// SIMATIC S7-200 project (STEP 7-Micro/WIN), CPU 224 CN REL 02.01

ORGANIZATION_BLOCK MAIN:OB1
TITLE=程序注释
BEGIN
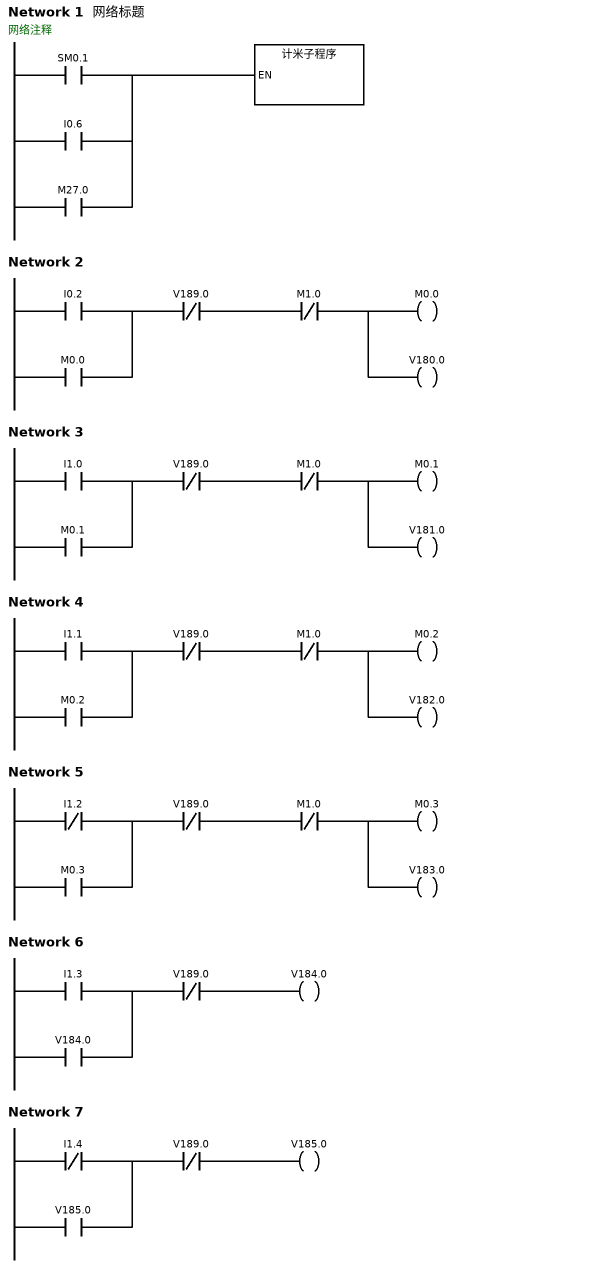
Network 1 // 网络标题
// 网络注释
LD     SM0.1
O      I0.6
O      M27.0
CALL   计米子程序:SBR0
Network 2
LD     I0.2
O      M0.0
AN     V189.0
AN     M1.0
=      M0.0
=      V180.0
Network 3
LD     I1.0
O      M0.1
AN     V189.0
AN     M1.0
=      M0.1
=      V181.0
Network 4
LD     I1.1
O      M0.2
AN     V189.0
AN     M1.0
=      M0.2
=      V182.0
Network 5
LDN    I1.2
O      M0.3
AN     V189.0
AN     M1.0
=      M0.3
=      V183.0
Network 6
LD     I1.3
O      V184.0
AN     V189.0
=      V184.0
Network 7
LDN    I1.4
O      V185.0
AN     V189.0
=      V185.0
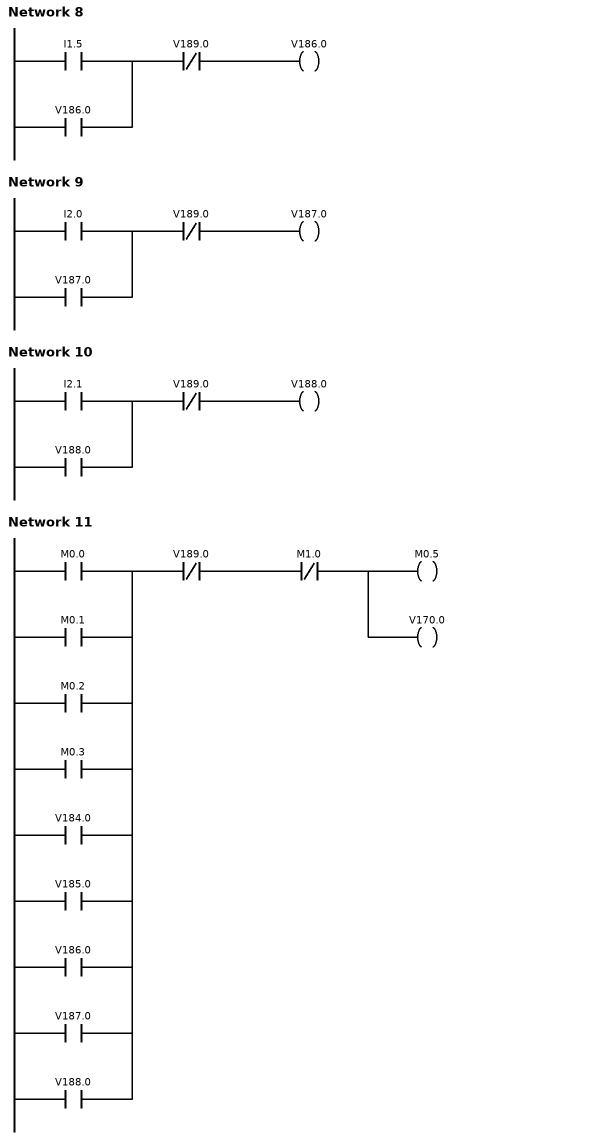
Network 8
LD     I1.5
O      V186.0
AN     V189.0
=      V186.0
Network 9
LD     I2.0
O      V187.0
AN     V189.0
=      V187.0
Network 10
LD     I2.1
O      V188.0
AN     V189.0
=      V188.0
Network 11
LD     M0.0
O      M0.1
O      M0.2
O      M0.3
O      V184.0
O      V185.0
O      V186.0
O      V187.0
O      V188.0
AN     V189.0
AN     M1.0
=      M0.5
=      V170.0
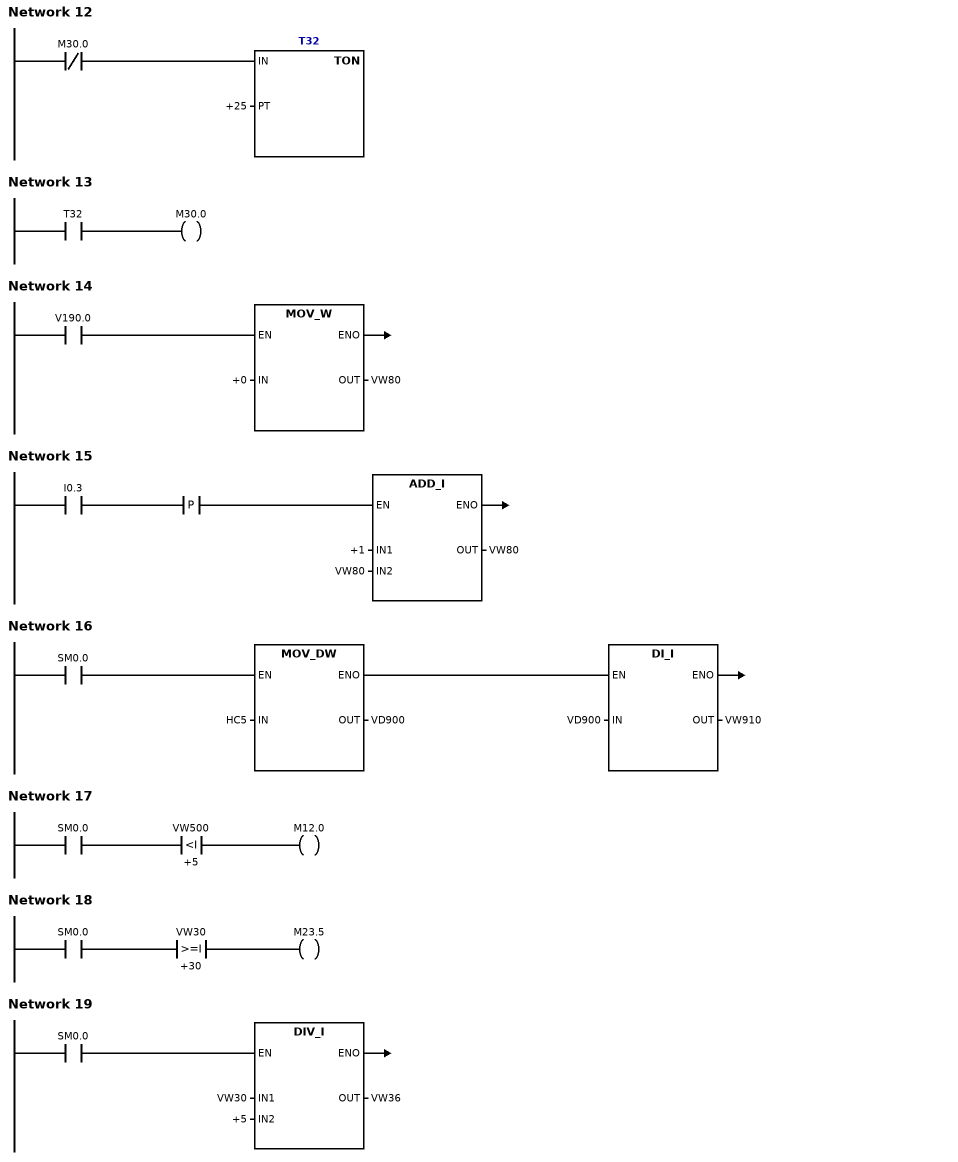
Network 12
LDN    M30.0
TON    T32, +25
Network 13
LD     T32
=      M30.0
Network 14
LD     V190.0
MOVW   +0, VW80
Network 15
LD     I0.3
EU
+I     +1, VW80
Network 16
LD     SM0.0
MOVD   HC5, VD900
AENO
DTI    VD900, VW910
Network 17
LD     SM0.0
AW<    VW500, +5
=      M12.0
Network 18
LD     SM0.0
AW>=   VW30, +30
=      M23.5
Network 19
LD     SM0.0
MOVW   VW30, VW36
/I     +5, VW36
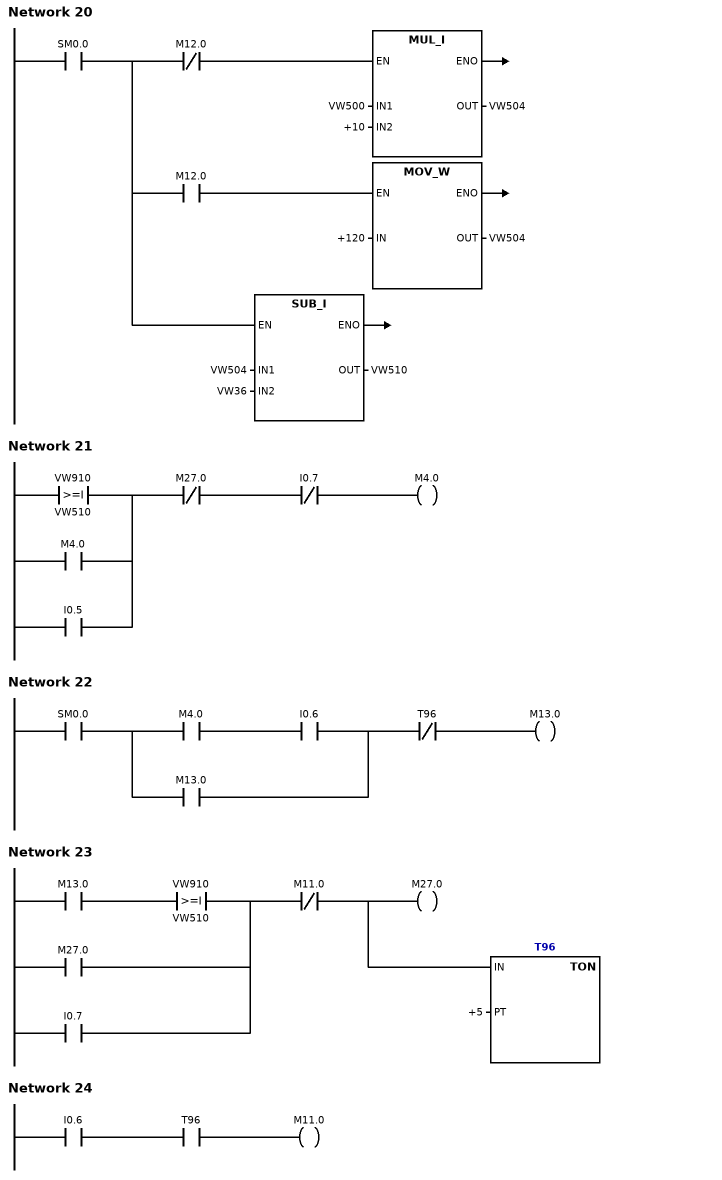
Network 20
LD     SM0.0
LPS
AN     M12.0
MOVW   VW500, VW504
*I     +10, VW504
LRD
A      M12.0
MOVW   +120, VW504
LPP
MOVW   VW504, VW510
-I     VW36, VW510
Network 21
LDW>=  VW910, VW510
O      M4.0
O      I0.5
AN     M27.0
AN     I0.7
=      M4.0
Network 22
LD     SM0.0
LD     M4.0
A      I0.6
O      M13.0
ALD
AN     T96
=      M13.0
Network 23
LD     M13.0
AW>=   VW910, VW510
O      M27.0
O      I0.7
AN     M11.0
=      M27.0
TON    T96, +5
Network 24
LD     I0.6
A      T96
=      M11.0
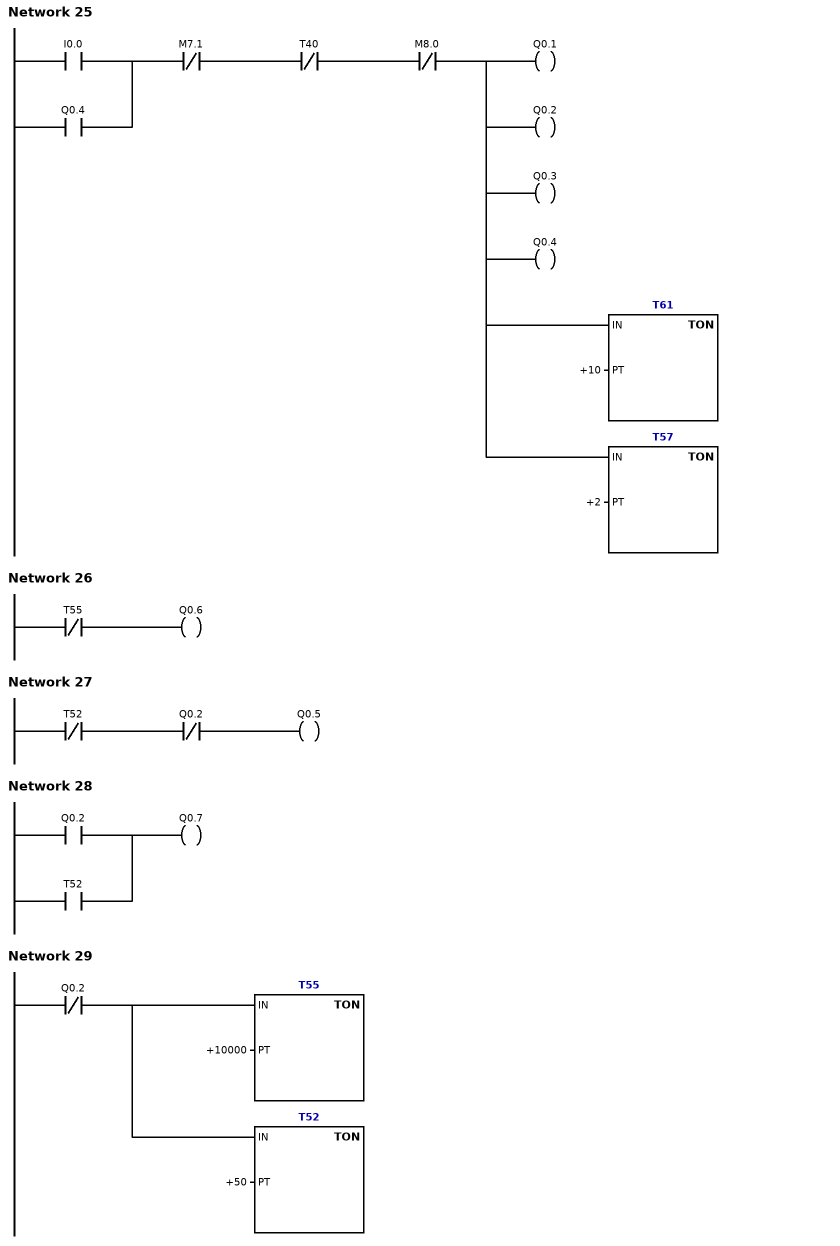
Network 25
LD     I0.0
O      Q0.4
AN     M7.1
AN     T40
AN     M8.0
=      Q0.1
=      Q0.2
=      Q0.3
=      Q0.4
TON    T61, +10
TON    T57, +2
Network 26
LDN    T55
=      Q0.6
Network 27
LDN    T52
AN     Q0.2
=      Q0.5
Network 28
LD     Q0.2
O      T52
=      Q0.7
Network 29
LDN    Q0.2
TON    T55, +10000
TON    T52, +50
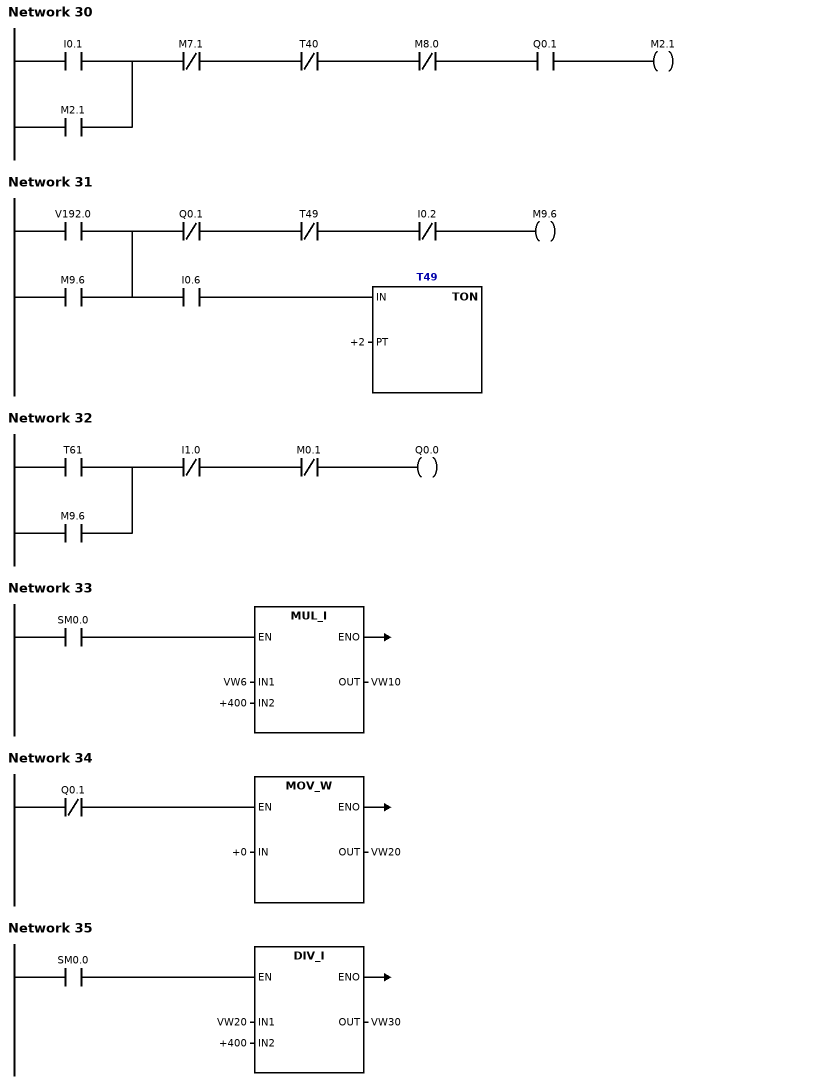
Network 30
LD     I0.1
O      M2.1
AN     M7.1
AN     T40
AN     M8.0
A      Q0.1
=      M2.1
Network 31
LD     V192.0
O      M9.6
LPS
AN     Q0.1
AN     T49
AN     I0.2
=      M9.6
LPP
A      I0.6
TON    T49, +2
Network 32
LD     T61
O      M9.6
AN     I1.0
AN     M0.1
=      Q0.0
Network 33
LD     SM0.0
MOVW   VW6, VW10
*I     +400, VW10
Network 34
LDN    Q0.1
MOVW   +0, VW20
Network 35
LD     SM0.0
MOVW   VW20, VW30
/I     +400, VW30
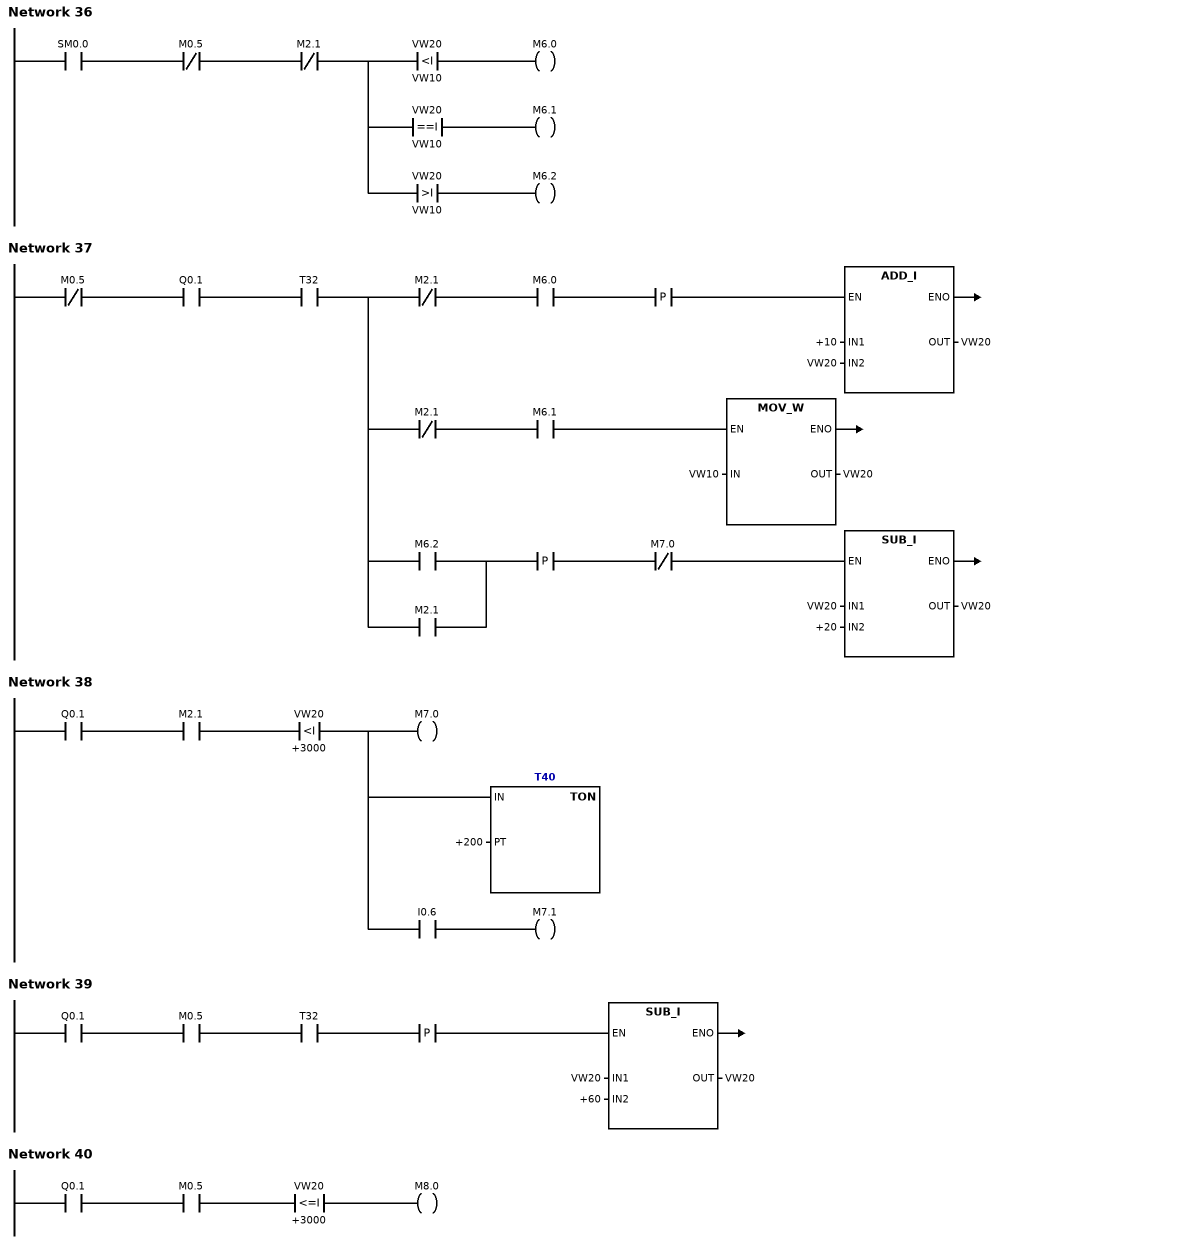
Network 36
LD     SM0.0
AN     M0.5
AN     M2.1
LPS
AW<    VW20, VW10
=      M6.0
LRD
AW=    VW20, VW10
=      M6.1
LPP
AW>    VW20, VW10
=      M6.2
Network 37
LDN    M0.5
A      Q0.1
A      T32
LPS
AN     M2.1
A      M6.0
EU
+I     +10, VW20
LRD
AN     M2.1
A      M6.1
MOVW   VW10, VW20
LPP
LD     M6.2
O      M2.1
ALD
EU
AN     M7.0
-I     +20, VW20
Network 38
LD     Q0.1
A      M2.1
AW<    VW20, +3000
=      M7.0
TON    T40, +200
A      I0.6
=      M7.1
Network 39
LD     Q0.1
A      M0.5
A      T32
EU
-I     +60, VW20
Network 40
LD     Q0.1
A      M0.5
AW<=   VW20, +3000
=      M8.0
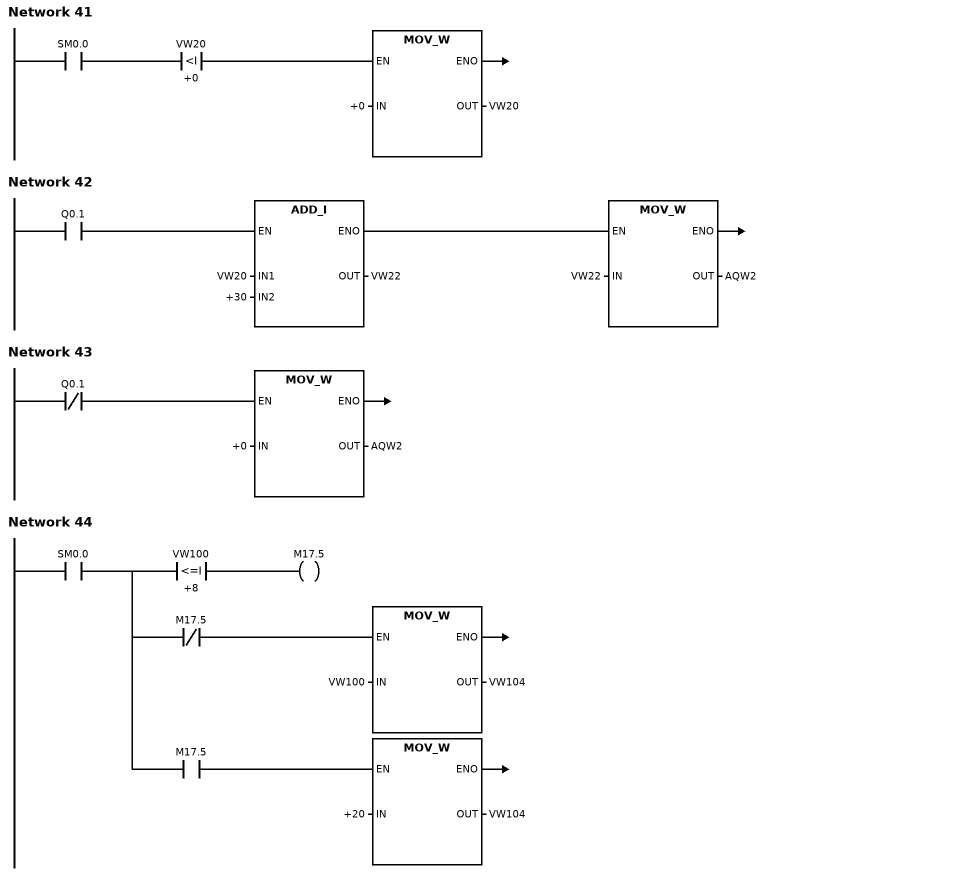
Network 41
LD     SM0.0
AW<    VW20, +0
MOVW   +0, VW20
Network 42
LD     Q0.1
MOVW   VW20, VW22
AENO
+I     +30, VW22
AENO
MOVW   VW22, AQW2
Network 43
LDN    Q0.1
MOVW   +0, AQW2
Network 44
LD     SM0.0
LPS
AW<=   VW100, +8
=      M17.5
LRD
AN     M17.5
MOVW   VW100, VW104
LPP
A      M17.5
MOVW   +20, VW104
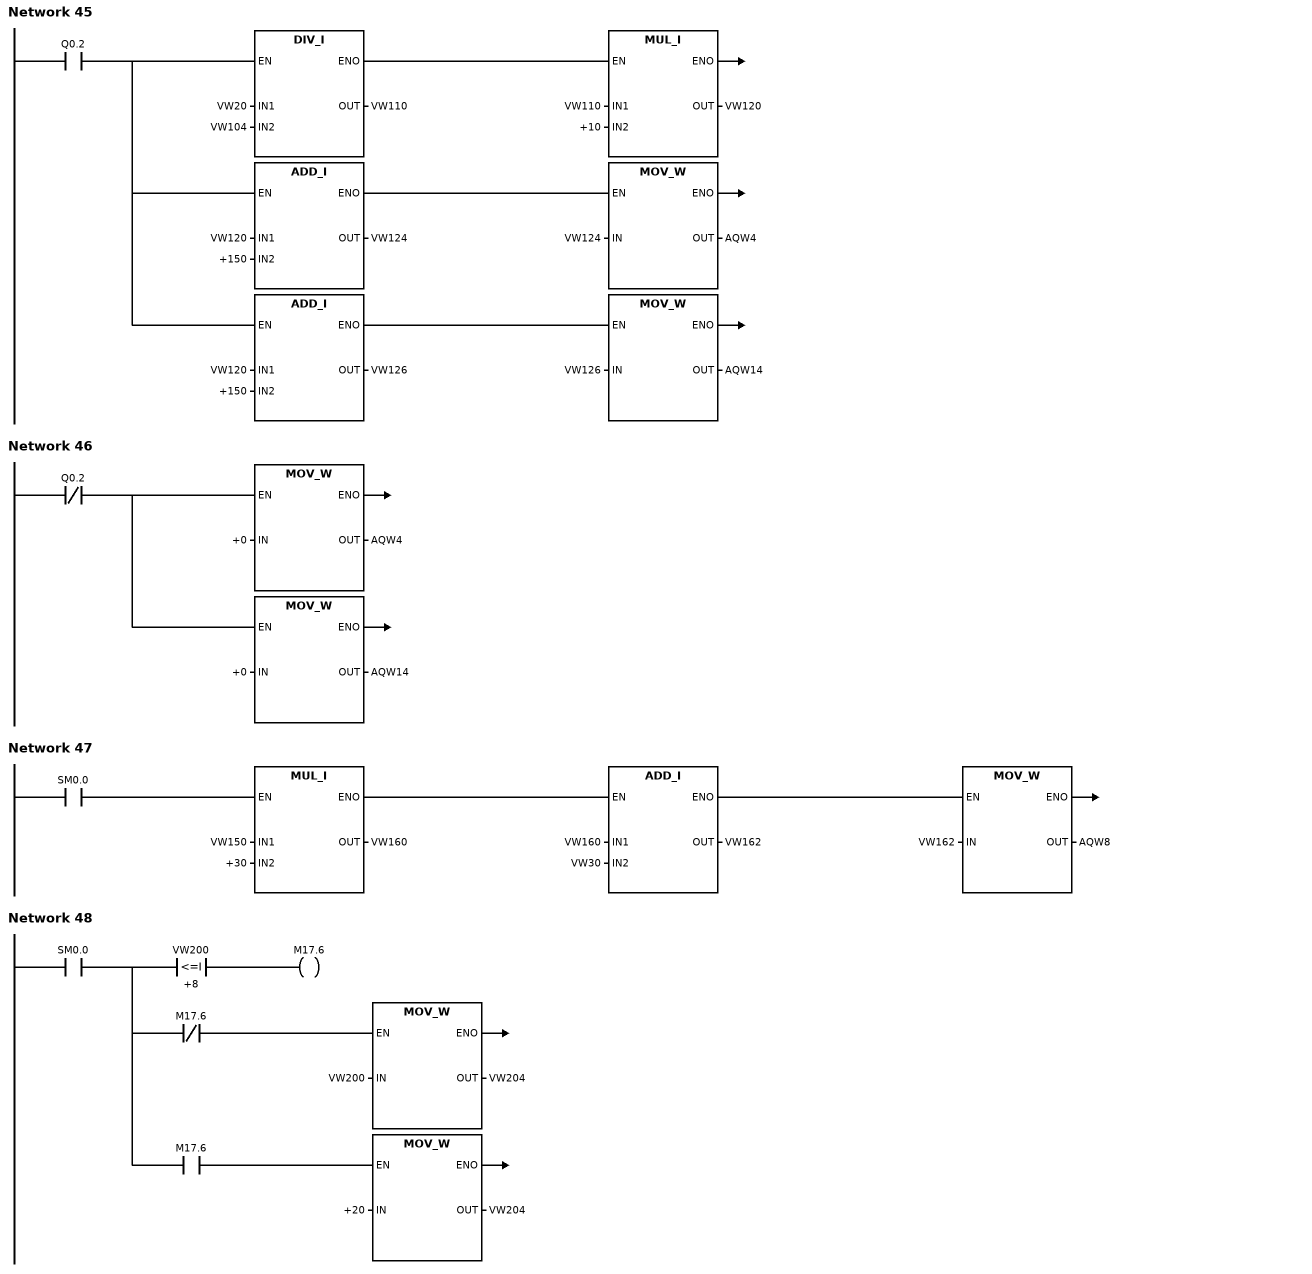
Network 45
LD     Q0.2
LPS
MOVW   VW20, VW110
AENO
/I     VW104, VW110
AENO
MOVW   VW110, VW120
*I     +10, VW120
LRD
MOVW   VW120, VW124
AENO
+I     +150, VW124
AENO
MOVW   VW124, AQW4
LPP
MOVW   VW120, VW126
AENO
+I     +150, VW126
AENO
MOVW   VW126, AQW14
Network 46
LDN    Q0.2
MOVW   +0, AQW4
MOVW   +0, AQW14
Network 47
LD     SM0.0
MOVW   VW150, VW160
AENO
*I     +30, VW160
AENO
MOVW   VW160, VW162
AENO
+I     VW30, VW162
AENO
MOVW   VW162, AQW8
Network 48
LD     SM0.0
LPS
AW<=   VW200, +8
=      M17.6
LRD
AN     M17.6
MOVW   VW200, VW204
LPP
A      M17.6
MOVW   +20, VW204
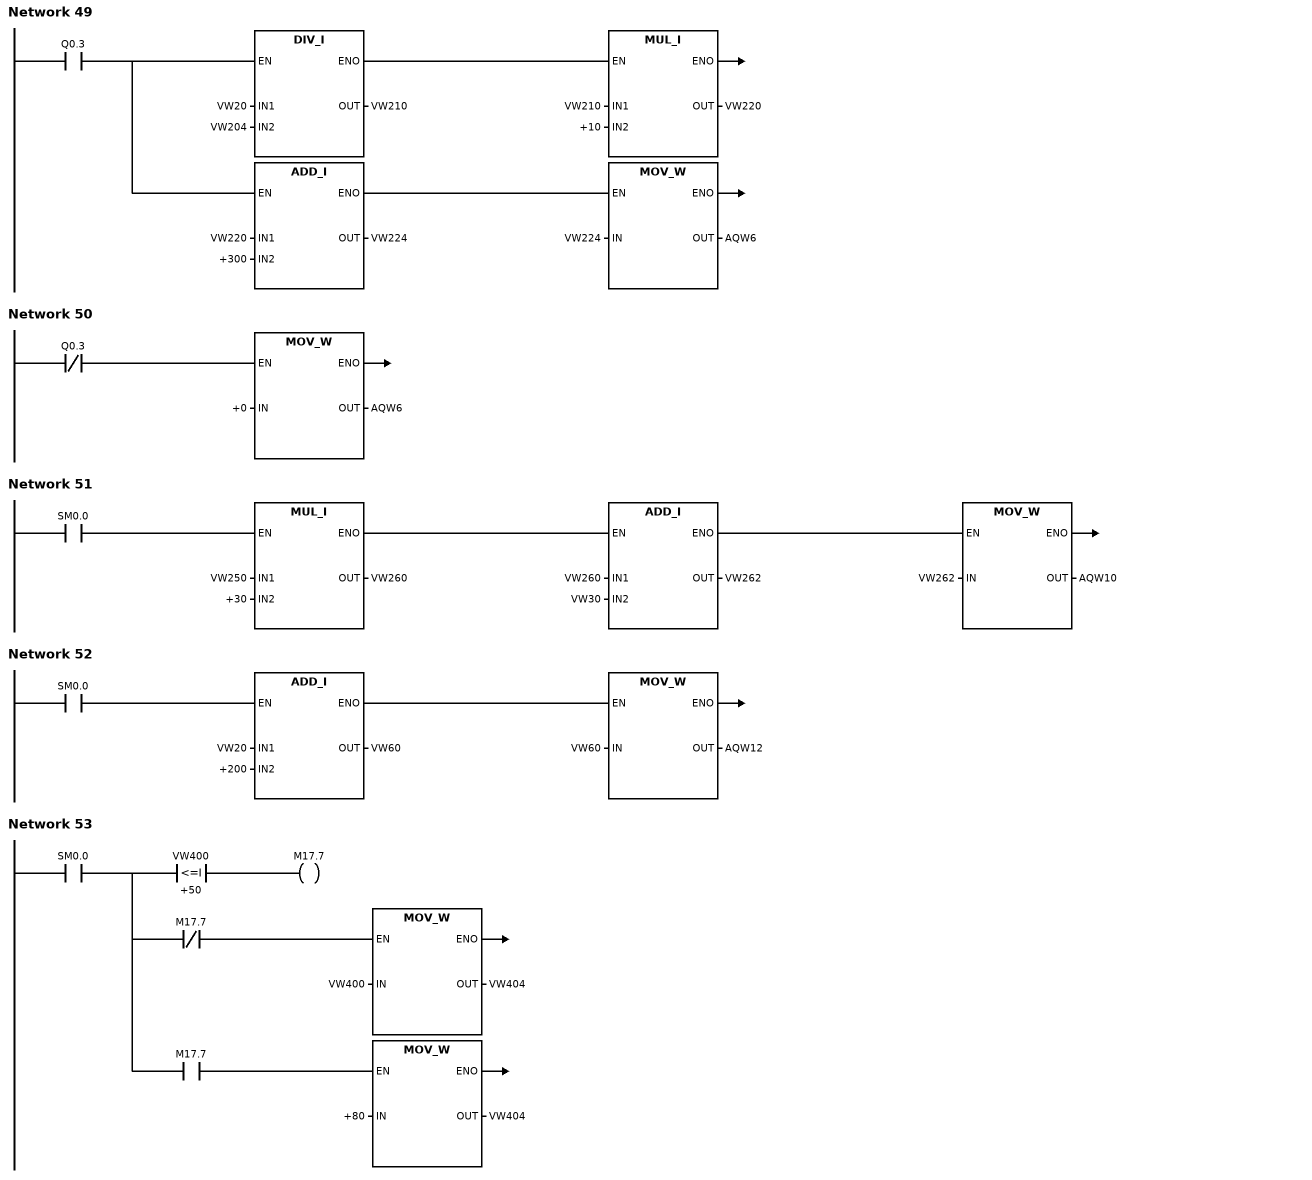
Network 49
LD     Q0.3
LPS
MOVW   VW20, VW210
AENO
/I     VW204, VW210
AENO
MOVW   VW210, VW220
*I     +10, VW220
LPP
MOVW   VW220, VW224
AENO
+I     +300, VW224
AENO
MOVW   VW224, AQW6
Network 50
LDN    Q0.3
MOVW   +0, AQW6
Network 51
LD     SM0.0
MOVW   VW250, VW260
AENO
*I     +30, VW260
AENO
MOVW   VW260, VW262
AENO
+I     VW30, VW262
AENO
MOVW   VW262, AQW10
Network 52
LD     SM0.0
MOVW   VW20, VW60
AENO
+I     +200, VW60
AENO
MOVW   VW60, AQW12
Network 53
LD     SM0.0
LPS
AW<=   VW400, +50
=      M17.7
LRD
AN     M17.7
MOVW   VW400, VW404
LPP
A      M17.7
MOVW   +80, VW404
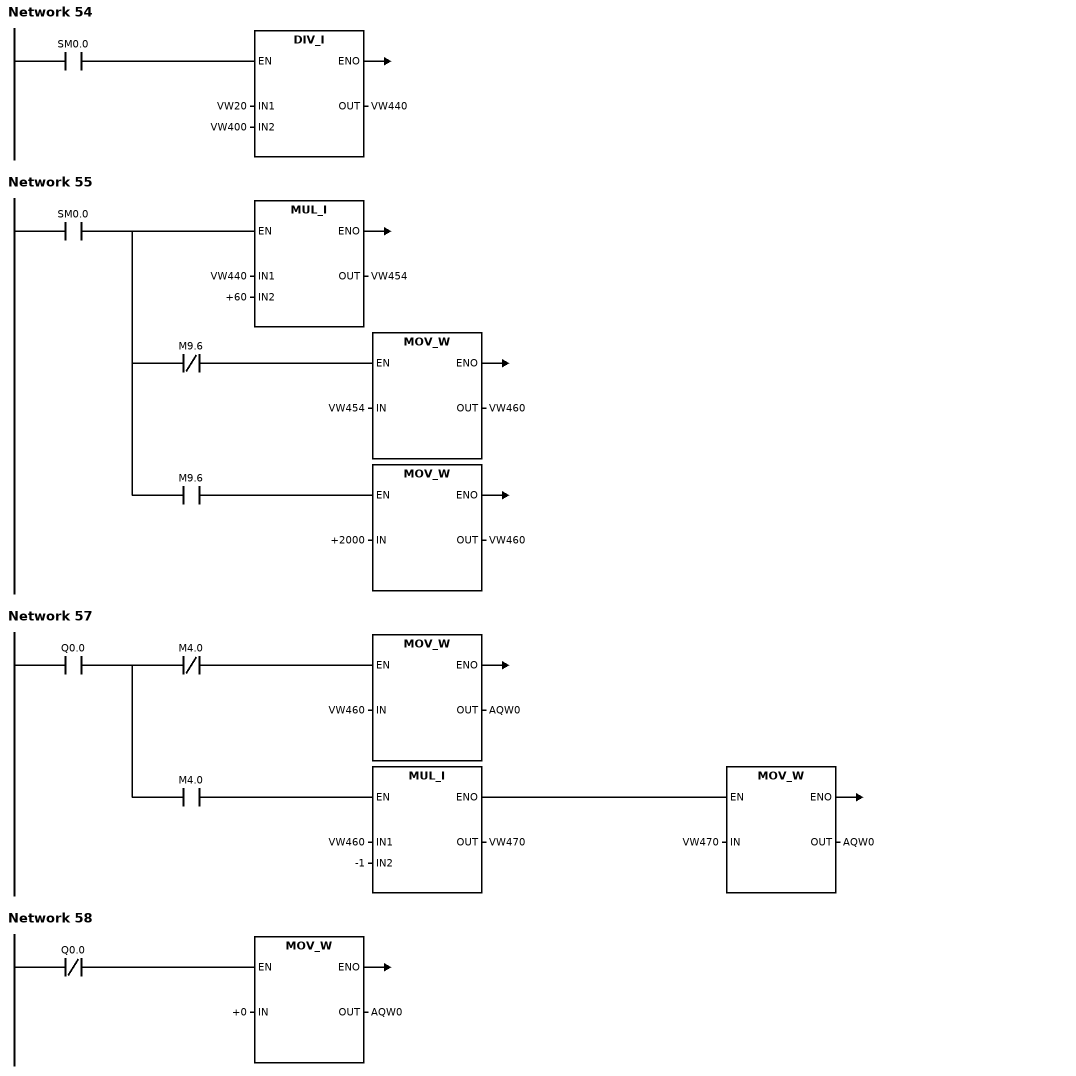
Network 54
LD     SM0.0
MOVW   VW20, VW440
/I     VW400, VW440
Network 55
LD     SM0.0
LPS
MOVW   VW440, VW454
*I     +60, VW454
AN     M9.6
MOVW   VW454, VW460
LPP
A      M9.6
MOVW   +2000, VW460
Network 57
LD     Q0.0
LPS
AN     M4.0
MOVW   VW460, AQW0
LPP
A      M4.0
MOVW   VW460, VW470
AENO
*I     -1, VW470
AENO
MOVW   VW470, AQW0
Network 58
LDN    Q0.0
MOVW   +0, AQW0
END_ORGANIZATION_BLOCK

SUBROUTINE_BLOCK 计米子程序:SBR0
TITLE=子程序注释
BEGIN
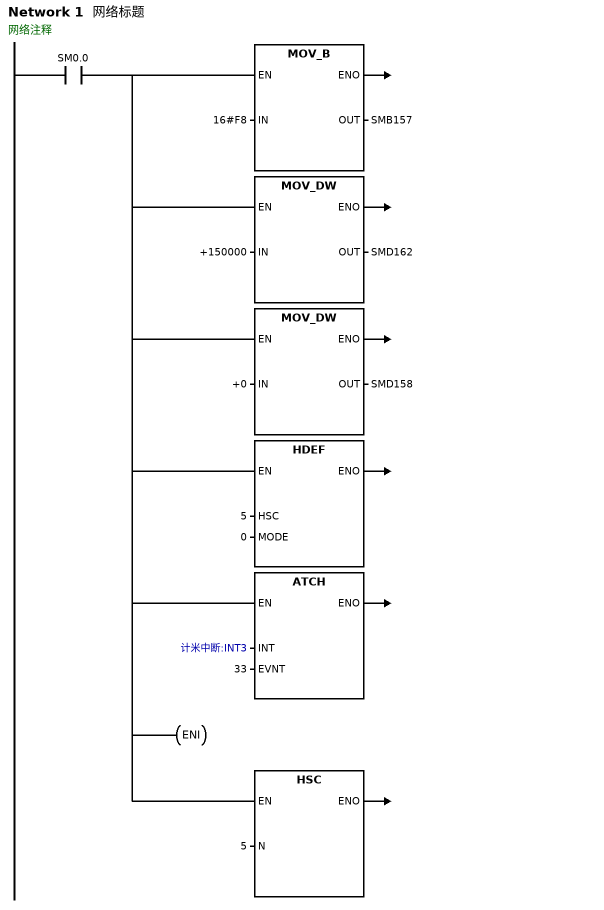
Network 1 // 网络标题
// 网络注释
LD     SM0.0
MOVB   16#F8, SMB157
MOVD   +150000, SMD162
MOVD   +0, SMD158
HDEF   5, 0
ATCH   计米中断:INT3, 33
ENI
HSC    5
END_SUBROUTINE_BLOCK

SUBROUTINE_BLOCK 放线:SBR1
TITLE=
BEGIN
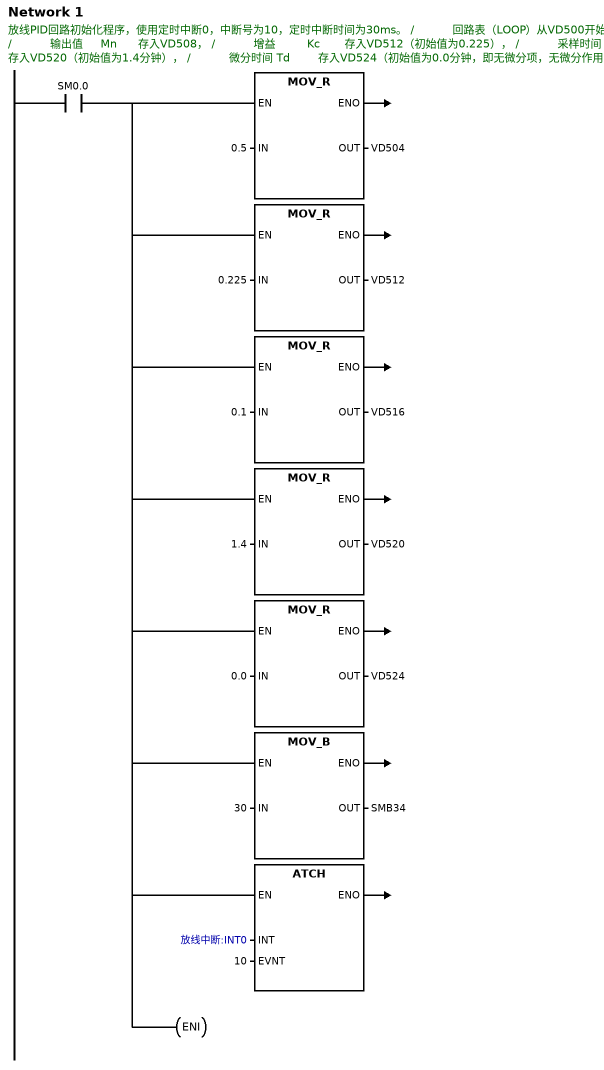
Network 1
//  放线PID回路初始化程序，使用定时中断0，中断号为10，定时中断时间为30ms。
//           回路表（LOOP）从VD500开始，
//           过程变量 PVn     存入VD500，
//           设定值     SPn     存入VD504（初始化为0.5），
//           输出值     Mn      存入VD508，
//           增益         Kc       存入VD512（初始值为0.225），
//           采样时间 Ts        存入VD516（初始值为0.1秒），
//           积分时间 Ti         存入VD520（初始值为1.4分钟），
//           微分时间 Td        存入VD524（初始值为0.0分钟，即无微分项，无微分作用）。
//     
//  
// 
LD     SM0.0
MOVR   0.5, VD504
MOVR   0.225, VD512
MOVR   0.1, VD516
MOVR   1.4, VD520
MOVR   0.0, VD524
MOVB   30, SMB34
ATCH   放线中断:INT0, 10
ENI
END_SUBROUTINE_BLOCK

SUBROUTINE_BLOCK 收线子程序:SBR2
TITLE=
BEGIN
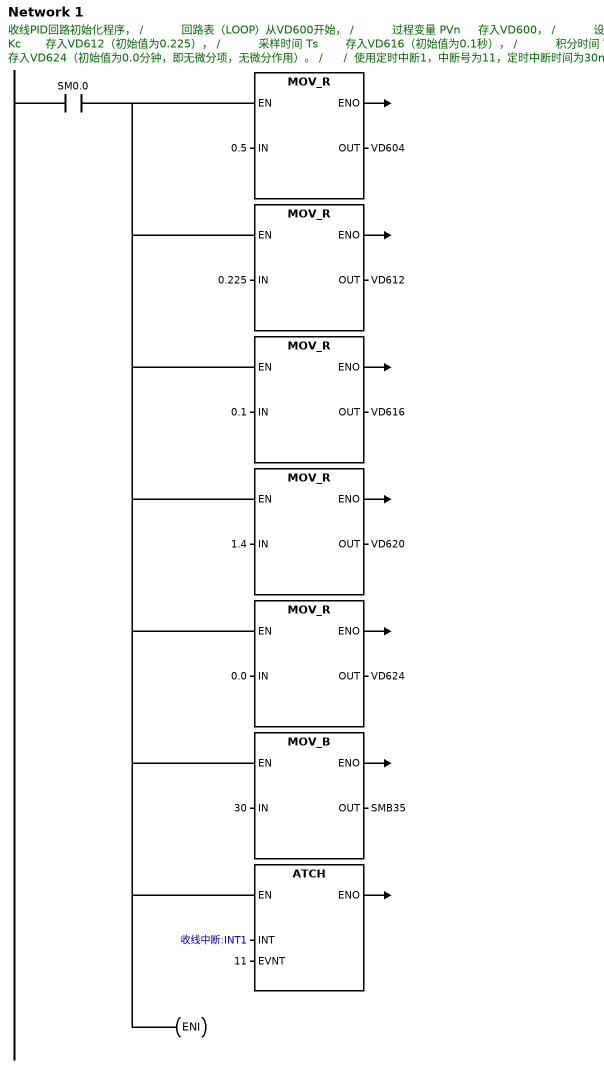
Network 1
//  收线PID回路初始化程序，
//           回路表（LOOP）从VD600开始，
//           过程变量 PVn     存入VD600，
//           设定值     SPn     存入VD604（初始化为0.5），
//           输出值     Mn      存入VD608，
//           增益         Kc       存入VD612（初始值为0.225），
//           采样时间 Ts        存入VD616（初始值为0.1秒），
//           积分时间 Ti         存入VD620（初始值为1.4分钟），
//           微分时间 Td        存入VD624（初始值为0.0分钟，即无微分项，无微分作用）。
//     
//  使用定时中断1，中断号为11，定时中断时间为30ms。
// 
LD     SM0.0
MOVR   0.5, VD604
MOVR   0.225, VD612
MOVR   0.1, VD616
MOVR   1.4, VD620
MOVR   0.0, VD624
MOVB   30, SMB35
ATCH   收线中断:INT1, 11
ENI
END_SUBROUTINE_BLOCK

INTERRUPT_BLOCK 放线中断:INT0
TITLE=中断程序注释
BEGIN
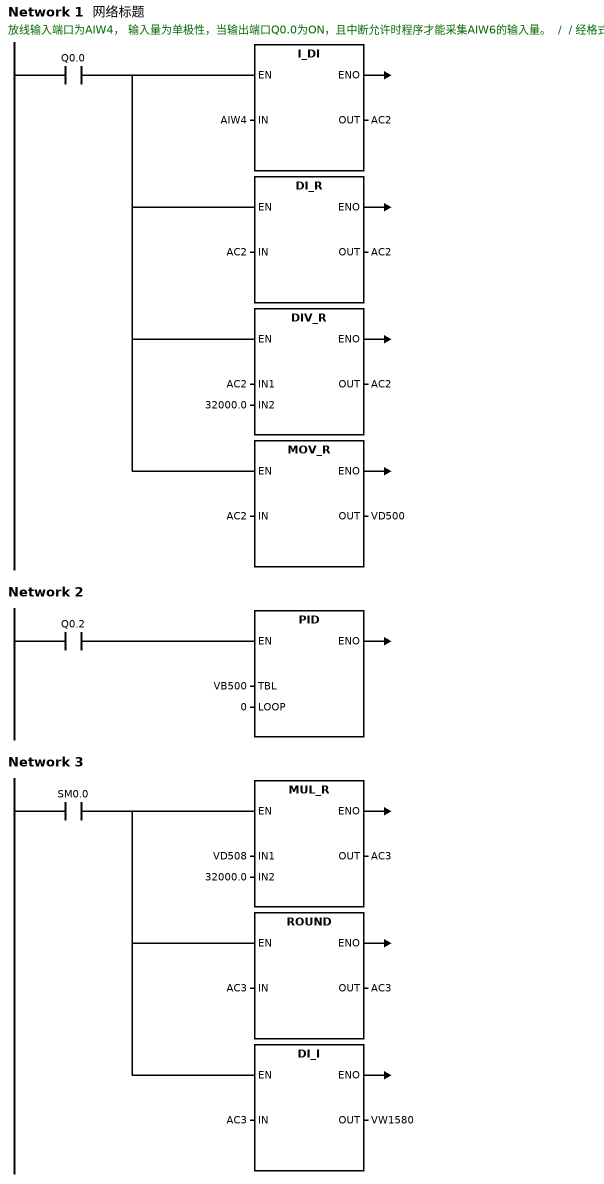
Network 1 // 网络标题
// 放线输入端口为AIW4， 输入量为单极性，当输出端口Q0.0为ON，且中断允许时程序才能采集AIW6的输入量。 
// 
// 经格式化后的输入过程变量存在VD500中  ，经反格式化后的变量存入VW1580。
LD     Q0.0
ITD    AIW4, AC2
DTR    AC2, AC2
/R     32000.0, AC2
MOVR   AC2, VD500
Network 2
LD     Q0.2
PID    VB500, 0
Network 3
LD     SM0.0
MOVR   VD508, AC3
*R     32000.0, AC3
ROUND  AC3, AC3
DTI    AC3, VW1580
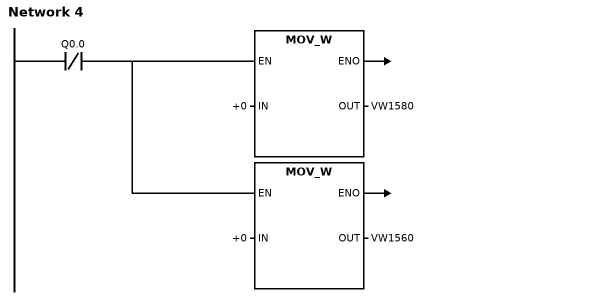
Network 4
LDN    Q0.0
MOVW   +0, VW1580
MOVW   +0, VW1560
END_INTERRUPT_BLOCK

INTERRUPT_BLOCK 收线中断:INT1
TITLE=
BEGIN
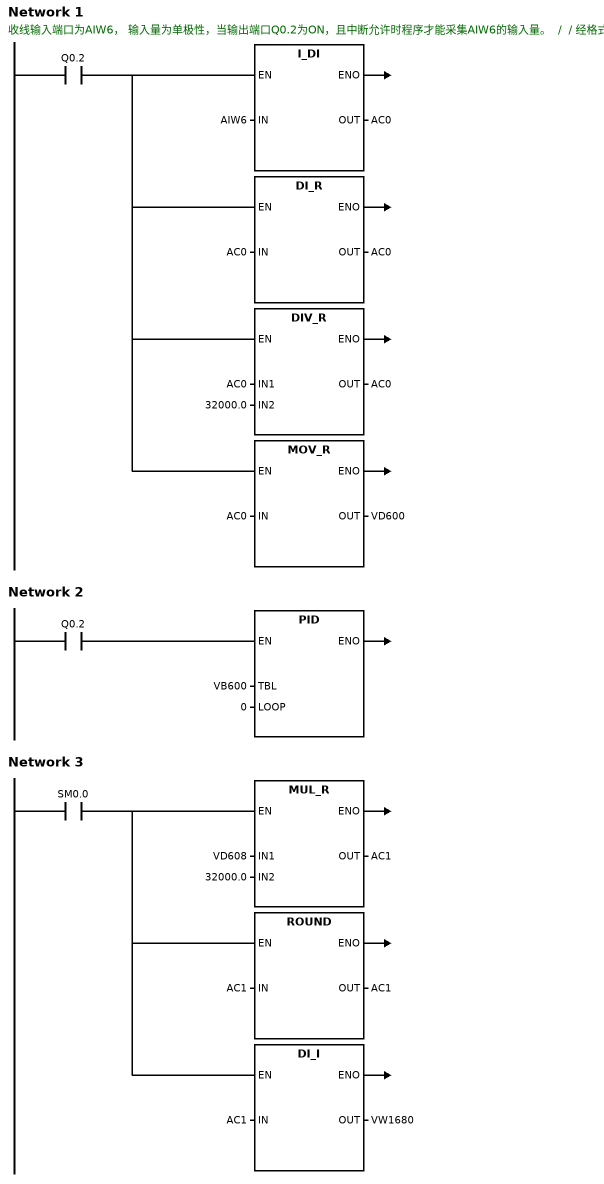
Network 1
// 收线输入端口为AIW6， 输入量为单极性，当输出端口Q0.2为ON，且中断允许时程序才能采集AIW6的输入量。 
// 
// 经格式化后的输入过程变量存在VD600中  ，经反格式化后的变量存入VW1680。
LD     Q0.2
ITD    AIW6, AC0
DTR    AC0, AC0
/R     32000.0, AC0
MOVR   AC0, VD600
Network 2
LD     Q0.2
PID    VB600, 0
Network 3
LD     SM0.0
MOVR   VD608, AC1
*R     32000.0, AC1
ROUND  AC1, AC1
DTI    AC1, VW1680
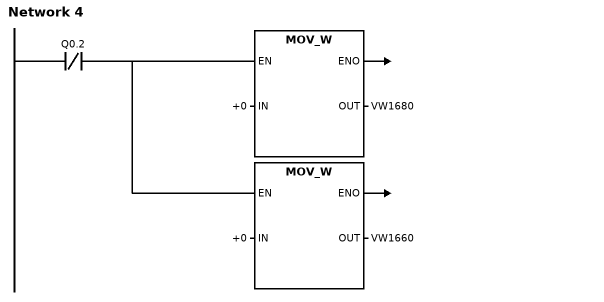
Network 4
LDN    Q0.2
MOVW   +0, VW1680
MOVW   +0, VW1660
END_INTERRUPT_BLOCK

INTERRUPT_BLOCK 计米中断:INT3
TITLE=
BEGIN
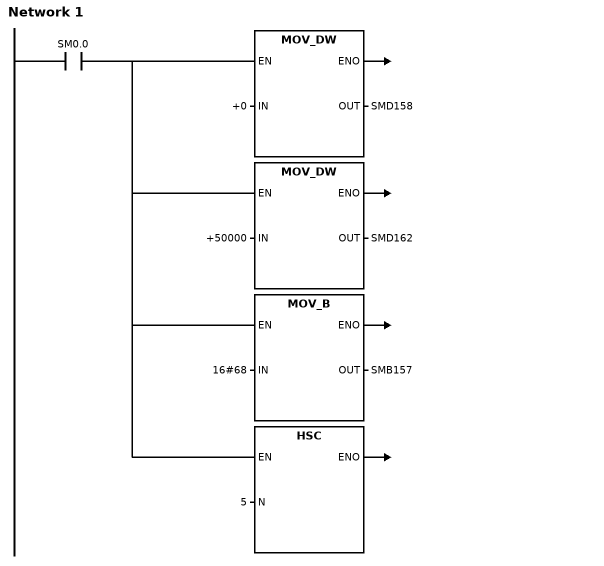
Network 1
LD     SM0.0
MOVD   +0, SMD158
MOVD   +50000, SMD162
MOVB   16#68, SMB157
HSC    5
END_INTERRUPT_BLOCK
